// TIA Portal V19 export
TYPE "LEXCHANGETRAY_typeTrayPosition"
// stored: Access Published
   STRUCT
      position : Word;   // 1:logistic 2: em1 4:em2 8:em5 16:em6
      logistic : Bool;   // 物流线
      EM1 : Bool;   // roller
      EM2 : Bool;   // constraintRoller
      EM6 : Bool;
      EM5 : Bool;
   END_STRUCT;
END_TYPE
